(* CODESYS project Meu projeto - PicK IN PLACE XYZ_.project

Project tree, tasks and I/O mapping:
  Device : CODESYS Control Win V3, 3S - Smart Software Solutions GmbH, order no. 305021, version 3.5.11.0
    application Application
      libraries: Standard, * (System)
      task MainTask (cyclic, interval t#20ms, priority 1) calls PLC_PRG
      program PLC_PRG [LD]
      global variables GVL
      function block FB_AUTOMAT [ST]
      Symbols
*)

// Device/Application/GVL
{attribute 'qualified_only'}
VAR_GLOBAL
	
  bAuto:BOOL;
   bBoxAtPlace:BOOL;
   bCLimit:BOOL;
   bDetected:BOOL;
   bEmergencyStop:BOOL;
   bManual:BOOL;
   bPartAtPlace:BOOL;
   bReset:BOOL;
   bStart:BOOL;
   bStop:BOOL;
    rX:REAL;
    rY:REAL;
    rZ:REAL;
	
bBoxConveyor:BOOL;
bBoxEmitter:BOOL;
bBoxRemover:BOOL;
bCplus:BOOL;
iCounter:INT;
bExitConveyor:BOOL;
bExitGreen:BOOL;
bExitRed:BOOL;
bExitYellow:BOOL;
bGrab:BOOL;
bPartConveyor:BOOL;
bPartEmitter:BOOL;
bResetLight:BOOL;
rSPX:REAL;
rSPY:REAL;
rSPZ:REAL;

bStartLight:BOOL;
bStopLight:BOOL;

END_VAR

// Device/Application/PLC_PRG
PROGRAM PLC_PRG
VAR
	FB_AUTOMAT_0: FB_AUTOMAT;
END_VAR

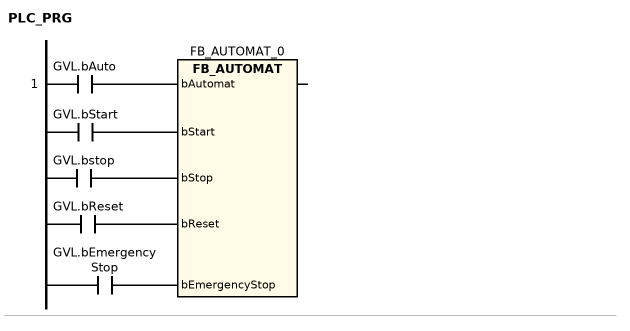
// NETWORK 1
FB_AUTOMAT_0(
    bAutomat := GVL.bAuto,
    bStart := GVL.bStart,
    bStop := GVL.bstop,
    bReset := GVL.bReset,
    bEmergencyStop := GVL.bEmergencyStop); // FB_AUTOMAT

END_PROGRAM

// Device/Application/FB_AUTOMAT
FUNCTION_BLOCK FB_AUTOMAT
VAR_INPUT
bAutomat:BOOL;
bStart:BOOL;
bStop:BOOL;
bReset:BOOL;
bEmergencyStop:BOOL;
END_VAR
VAR_OUTPUT
END_VAR
VAR
block:BOOL;
Work:BOOL;
step:INT;
step_part:INT;
step_box:INT;
step_exit:INT;
BOX_TRIG:F_TRIG;
END_VAR


///////**********************************************************************************************************///////
                  //Sistema Pick in place - manipulador de caixas - 3 Eixos//
	
/////////////*****************************************************************************************////////



///////Rotina sequencial ////////

BOX_TRIG(CLK:=GVL.bBoxAtPlace);
IF NOT block THEN

CASE step OF
    1:
        step_part:=1;
        step_part:=1;
        step:= 2;
		
  	2:     IF NOT GVL.bBoxAtPlace AND NOT GVL.bPartAtPlace THEN
           step:=3;
		   
	   END_IF
	   
    3:
        GVL.rSPX:=8;
        GVL.rSPY:=5.6;
        IF GVL.rX>7.9 AND GVL.rY>5.5 THEN
           step:=4;
       END_IF
	   
     4:  GVL.rSPZ:= 5;
        IF GVL.bDetected THEN
           GVL.bGrab:=TRUE;
           step:=5;
       END_IF
	   
    5:
        GVL.rSPZ:=0;
        step_part:=1;
        IF GVL.rZ<0.1 THEN
           step:= 6;
        END_IF

	6: 

	GVL.rSPX:=3.3;
	GVL.rSPY:=6.7;
	
	IF GVL.rX>3.2 AND GVL.rY>6.6 THEN
    	step:=7;
	END_IF
	
	7:
	
	GVL.rSPZ:=10;
	IF GVL.rZ>9.9 THEN
    step:=8;
	END_IF
	
	8:
	
	GVL.bGrab:=FALSE;
	GVL.rSPZ:=0;
	IF GVL.rZ<0.1 THEN
    step:=9;
	END_IF
	
	9:
	GVL.rSPX:=8;
	GVL.rSPY:=5.6;
	IF GVL.rX>7.9 AND GVL.rY>5.5 THEN
    step:=10;
	END_IF
	
	 10:

     GVL.rSPZ:=4.8;
     IF GVL.bDetected THEN
          GVL.bGrab:=TRUE;
          step:=11;
    END_IF
	
	11:
	
     GVL.rSPZ:=0;
     step_part:=1;
    IF GVL.rZ<0.1 THEN
          step:=12;
    END_IF
	
	12:
	
     GVL.rSPX:=3.3;
     GVL.rSPY:=3.1;
     IF GVL.rX<3.4 AND GVL.rY<3.2 THEN
          step:=13;
    END_IF
	
	13:
	
    GVL.rSPZ:=10;
    IF GVL.rZ>9.9 THEN
          step:=14;
    END_IF
	
	14:
	 
     GVL.bGrab:=FALSE;
     GVL.rSPZ:=0;
     IF GVL.rz<0.01 THEN
          step:=15;
    END_IF
	

15:

    GVL.rSPX:=8;
    GVL.rSPY:=5.6;
    IF GVL.rX>7.9 AND GVL.rY>5.5 THEN
        step:=16;
    END_IF
	
16:

    GVL.rSPZ:=4.8;
    IF GVL.bDetected THEN
        GVL.bGrab:=TRUE;
        step:=17;
    END_IF
	
17:
    GVL.rSPZ:=0;
    step_part:=1;
    IF GVL.rZ<0.1 THEN
        step:=18;
    END_IF
	
	
18:

    GVL.rSPX:=3.3;
    GVL.rSPY:=5;
    GVL.bCplus:=TRUE;
    IF GVL.rX<3.4 AND GVL.rY<5.1 AND GVL.bCLimit THEN
        step:=19;
    END_IF
	
19:

    GVL.rSPZ:=5.7;
    IF GVL.rZ>5.6 THEN
        step:=20;
    END_IF
	
20:

    GVL.bGrab:=FALSE;
    GVL.rSPZ:=0;
    IF GVL.rZ<0.01 THEN
        step:=21;
        GVL.bCplus:=FALSE;
    END_IF
	
21:

    step_box:=1;
    step:=22;
    GVL.iCounter:=GVL.iCounter+1;         /// Contagem de caixas
	
22:

    IF Work THEN
        step:=1;
    ELSE
        step:=0;
    END_IF
	
END_CASE
END_IF

/////Sub-rotina  de esteira de baixo////

CASE step_part OF
    1:
        GVL.bPartConveyor:=TRUE;
        IF NOT GVL.bPartAtPlace THEN
            step_part:=2;
        END_IF
		
	2:
        GVL.bPartConveyor:=FALSE;
		
END_CASE


////////////////////////////////////////////////
///sub - rotina esteira de cima /////////

CASE step_box OF
	
	1:

        GVL.bBoxConveyor:=TRUE;
        step_exit:=1;
        IF BOX_TRIG.Q THEN
            step_box:=2;
            step_exit:=2;
        END_IF
		
	2:
        GVL.bBoxConveyor:=FALSE;
		
END_CASE

//////////////////////////////////////////////////////////

CASE step_exit OF
	
1:
    GVL.bExitConveyor:=TRUE;
2:
     GVL.bExitConveyor:=FALSE;
END_CASE

///////////////////////////////////////////////////////////

////* Acionamento do sistema ///////////////////////


IF bStart AND bAutomat AND NOT block AND GVL.bBoxAtPlace THEN
	Work:=TRUE;
	step:=1;
	step_part:=1;
	step_box:=1;
END_IF


IF bStart AND bAutomat AND NOT block AND NOT GVL.bBoxAtPlace THEN
	Work:=TRUE;
	step:=2;
	
END_IF

IF NOT bStop THEN
	Work:=FALSE;
	step:=0;
END_IF



/////////////Rotina de emergência////////////


IF NOT bEmergencyStop THEN
    Work:=FALSE;
    block:=TRUE;
    // step:=0;
    step_part:=0;
    step_box:=0;
    step_exit:=0;
    //GVL.rSPX:=0;
    //GVL.rSPY:=0;
    GVL.rSPZ:=0;
    GVL.bBoxConveyor:=FALSE;
    GVL.bPartConveyor:=FALSE;
END_IF


IF bEmergencyStop AND bReset THEN
    block:=FALSE;
END_IF

GVL.bResetLight:=block;
GVL.bStartLight:=Work;

/////////////////////////////////////qq

/////sinalização///////////////

GVL.bStopLight:=NOT Work;
GVL.bExitGreen:=Work;
GVL.bExitRed:=NOT Work;
GVL.bExitYellow:=block;

END_FUNCTION_BLOCK
